FUNCTION_BLOCK ABSTRACT FB_HasTaskInfo
VAR
	_PlcTaskInfo	: PlcTaskSystemInfo;
	_attempts	: UINT;
END_VAR

{attribute 'monitoring':='call'}
PROPERTY TaskInfo : REFERENCE TO PlcTaskSystemInfo
GET
VAR
	taskIndex	: DINT;
END_VAR
IF _plcTaskInfo.CycleTime = 0 THEN
	taskIndex := Tc2_System.GETCURTASKINDEXEX();
	IF taskIndex <> 0 THEN
		_PlcTaskInfo := _TaskInfo[taskindex];
	END_IF
END_IF

TaskInfo REF= _PlcTaskInfo;
END_GET
END_PROPERTY

END_FUNCTION_BLOCK

(* stored: Version 1.1.0.1, ProductVersion 3.1.4024.13
   POU FB_HasTaskInfo: Id {90620e8f-2928-015b-1ab1-9c3efa46279c}, SpecialFunc None
   Property TaskInfo: Id {bf63dea1-0cf1-00ee-1958-66e2577ef95f}
   Get Get: Id {fc727187-ae1f-07d1-141e-4eab00933cc9} *)
